// TIA Portal V16 export
// export: Created 2023-03-29T11:03:47.4049579Z, ExportSetting WithDefaults, DisplayName Totally Integrated Automation Portal, DisplayVersion V16 Update 6, DisplayName TIA Portal Version Control Interface, DisplayVersion V16 Update 2, DisplayName TIA Portal Openness, DisplayVersion V16 Update 6, DisplayName STEP 7 Professional, DisplayVersion V16 Update 6, DisplayName STEP 7 Safety, DisplayVersion V16, DisplayName WinCC Advanced, DisplayVersion V16 Update 6
TYPE "stt_OB82"
// stored: IsFailsafeCompliant false
   STRUCT
      ErrorTimestamp : DTL;   // //time error occurs
      IO_State : Word;   // //Contains the I/O status of the diagnostics-capable module.
      LADDR : HW_ANY;   // //HW-ID
      Channel : UInt;   // //Channel number
      MultiError : Bool;   // //= 1, if there is more than one error
   END_STRUCT;
END_TYPE
